(* CoDeSys 2.3.9.35 project: Exercício3.pro *)
(* Author: Altus *)
(* Libraries: DU35x.lib 7.7.11 15:59:13, Navigation.lib 15.7.11 10:06:00, SysLibTargetVisu.lib 26.11.08 09:53:28, Standard.lib 26.11.08 09:46:20, Iecsfc.lib 26.11.08 09:46:14, SYSLIBCALLBACK.LIB 26.11.08 09:53:30 *)

(* PLC configuration (modules and I/O channels)
Configuração do CP [Root] node -1, in %IB0 out %QB0
  Comunicação [Comunica] node 0, in %IB0 out %QB0
    COM1 [COM1] node 0, in %IB0 out %QB0 {BaudRate = 115200; Paridade = Sem Paridade; StopBits = 1 Stop Bit; Modem = Sem RTS/CTS; Delay = 5}
      MToolIEC [Codesys] node 0, in %IB0 out %QB0
    COM2 [COM2] node 1, in %IB0 out %QB0 {BaudRate = 115200; Paridade = Sem Paridade; StopBits = 1 Stop Bit; Modem = Sem RTS/CTS; Delay = 5}
      Desabilitada [Desabilitado485] node 0, in %IB0 out %QB0
  Barramento [Barramento] node 1, in %IB0 out %QB0
    Entradas [Entradas] node 0, in %IB0 out %QB0
      Entradas Digitais 0 [Entradas0] node 0, in %IW0 out %QB0
        I00 AT %IX0.0 [BitInput] I0.0
        I01 AT %IX0.1 [BitInput] I0.1
        I02 AT %IX0.2 [BitInput] I0.2
        I03 AT %IX0.3 [BitInput] I0.3
        I04 AT %IX0.4 [BitInput] I0.4
        I05 AT %IX0.5 [BitInput] I0.5
        I06 AT %IX0.6 [BitInput] I0.6
        I07 AT %IX0.7 [BitInput] I0.7
        I08 AT %IX0.8 [BitInput] I0.8
      Entradas Digitais 1 [Entradas1] node 0, in %IW1 out %QB0
        I10 AT %IX1.0 [BitInput] I1.0
        I11 AT %IX1.1 [BitInput] I1.1
        I12 AT %IX1.2 [BitInput] I1.2
        I13 AT %IX1.3 [BitInput] I1.3
        I14 AT %IX1.4 [BitInput] I1.4
        I15 AT %IX1.5 [BitInput] I1.5
        I16 AT %IX1.6 [BitInput] I1.6
        I17 AT %IX1.7 [BitInput] I1.7
        I18 AT %IX1.8 [BitInput] I1.8
      Entradas Digitais 2 [Entradas2] node 0, in %IW2 out %QB0
        I20 AT %IX2.0 [BitInput] I2.0
        I21 AT %IX2.1 [BitInput] I2.1
      Entradas Analógicas [EntradaAnalogica] node 0, in %IW4 out %QB0
        AI0 AT %IW4 [WordInput] AI0 {TipoAnalogica = Channel Disable; FiltroAnalogica = Filter 0 - AI=2ms  / AV=90ms; FundoEscala = 0}
        AI1 AT %IW5 [WordInput] AI1 {TipoAnalogica = Channel Disable; FiltroAnalogica = Filter 0 - AI=2ms  / AV=90ms; FundoEscala = 0}
        AI2 AT %IW6 [WordInput] AI2 {TipoAnalogica = Channel Disable; FiltroAnalogica = Filter 0 - AI=2ms  / AV=90ms; FundoEscala = 0}
        AI3 AT %IW7 [WordInput] AI3 {TipoAnalogica = Channel Disable; FiltroAnalogica = Filter 0 - AI=2ms  / AV=90ms; FundoEscala = 0}
      Entradas Rápidas [EntradasRapidas] node 1, in %IB16 out %QB0
        Bloco 0 [Bloco0] node 0, in %IB16 out %QB0
          Desabilitado [DesabilitadoBloco0] node 0, in %IB16 out %QB0
        Bloco 1 [Bloco1] node 1, in %IB16 out %QB0
          Desabilitado [DesabilitadoBloco1] node 0, in %IB16 out %QB0
        Entrada Configuravél Bloco 0 [EntradaConfiBloco0] node 2, in %IB16 out %QB0
          Contador 0 [EntradaConfContador0] node 0, in %IB16 out %QB0 {EntradaConfiguravelContador = Disable}
        Entrada Configuravél Bloco 1 [EntradaConfiBloco1] node 3, in %IB16 out %QB0
          Contador 2 [EntradaConfContador2] node 0, in %IB16 out %QB0 {EntradaConfiguravelContador = Disable}
    Saídas [Saidas] node 1, in %IB13 out %QB0
      Saídas Digitais 0 [Saidas0] node 0, in %IW0 out %QW0
        Q00 AT %QX0.0 [BitOutput] Q0.0
        Q01 AT %QX0.1 [BitOutput] Q0.1
        Q02 AT %QX0.2 [BitOutput] Q0.2
        Q03 AT %QX0.3 [BitOutput] Q0.3
        Q04 AT %QX0.4 [BitOutput] Q0.4
        Q05 AT %QX0.5 [BitOutput] Q0.5
        Q06 AT %QX0.6 [BitOutput] Q0.6
        Q07 AT %QX0.7 [BitOutput] Q0.7
      Saídas Digitais 1 [Saidas1] node 0, in %IW0 out %QW1
        Q10 AT %QX1.0 [BitOutput] Q1.0
        Q11 AT %QX1.1 [BitOutput] Q1.1
        Q12 AT %QX1.2 [BitOutput] Q1.2
        Q13 AT %QX1.3 [BitOutput] Q1.3
        Q14 AT %QX1.4 [BitOutput] Q1.4
        Q15 AT %QX1.5 [BitOutput] Q1.5
        Q16 AT %QX1.6 [BitOutput] Q1.6
        Q17 AT %QX1.7 [BitOutput] Q1.7
      Saídas Analógicas [SaidaAnalogica] node 0, in %IW0 out %QW3
        AO0 AT %QW3 [WordOutput] AO0 {TipoAnalogica = Channel Disable; FundoEscala = 0}
        AO1 AT %QW4 [WordOutput] AO1 {TipoAnalogica = Channel Disable; FundoEscala = 0}
      Saídas Rápidas [SaidasRapidas] node 1, in %IB0 out %QB10
        Saída Rápida 0 Desabilitada [DesabilitadoF0] node 0, in %IB0 out %QB10
        Saída Rápida 1 Desabilitada [DesabilitadoF1] node 1, in %IB0 out %QB10
      Saídas Comum de Contador [SaidasContador] node 2, in %IB0 out %QB10
        Saída do Bloco 0 Desabilitada [DesabilitadoSaidaBloco0] node 0, in %IB0 out %QB10
        Saída do Bloco 1 Desabilitada [DesabilitadoSaidaBloco1] node 1, in %IB0 out %QB10
  Eventos Externos [Eventos] node 2, in %IB13 out %QB6
    Evento Temporizado [TimerEvent] node 0, in %IB13 out %QB6 {Intervalo = 10}
*)

(* Task configuration *)
TASK PRINCIPAL (PRIORITY := 1, INTERVAL := T#1ms);
	PLC_PRG();
END_TASK
TASK NAVIGATION (PRIORITY := 1, INTERVAL := T#20ms);
	NAVEGA();
END_TASK
TASK VISUALIZATION (PRIORITY := 1, INTERVAL := T#500ms);
	MAINTARGETVISU_PAINT_CODE
END_TASK
TASK KEYBOARD_USAGE (PRIORITY := 1, INTERVAL := T#20ms);
	MAINTARGETVISU_INPUT_CODE
END_TASK

(* POU PLC_PRG, LD *)
(*Elabore um programa que produza uma rampa de tensão analógica para acionamento de um sistema partida e parada suaves de um motor (com um
sistema analógico com TCA785, por exemplo). Ao ser acionado um botão denominado LIGA no painel da IHM do CP, deve ser gerada uma rampa de 0V
a 10V na saída analógica, e de 10V a 0V ao ser acionado um botão denominado DESLIGA. O tempo de subida deve ser de 10s e tempo de descida de 
7s. Exiba o valor do percentual de potência na IHM. A rampa deve ter pelo menos 100 pontos de resolução. Prever o acionamento de uma saída 
digital no estado de potência zero e outra saída digital no estado de potência máxima. Exiba o valor de tensão de saída na IHM, de forma 
numérica e de forma gráfica (gráfico de tendência, por exemplo). Usar a escala apropriada (duas casa decimais) e com indicação de unidade.
*)

PROGRAM PLC_PRG
VAR
	LIG: BOOL;
	DES: BOOL;
	S1 AT %QX1.0: BOOL;
	S2 AT %QX1.1: BOOL := 1;
	AN AT %QW3: WORD;
	TS: TIME := T#10s;
	TD: TIME := T#7s;
	T1: TOF;
	T2: TOF;
	DESC: TIME;
	SUBI: TIME;
	BD1: F_TRIG;
	BD2: F_TRIG;
	BSS1: R_TRIG;
	BSS2: R_TRIG;
	BD: R_TRIG;
	BL: R_TRIG;
	M1: BOOL;
	M2: BOOL := 1;
	M3: BOOL;
	M4: BOOL;
	M5: BOOL;
	TR: WORD;
	SUBTR: REAL;
	SUBWORD: WORD;
	ANR: REAL;
	POT: REAL;
END_VAR
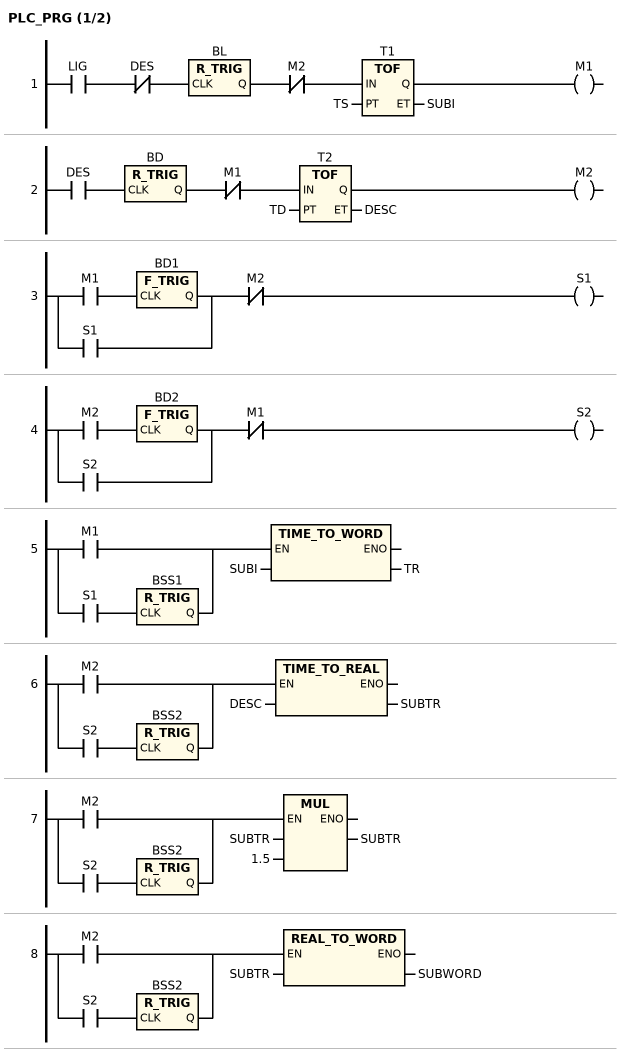
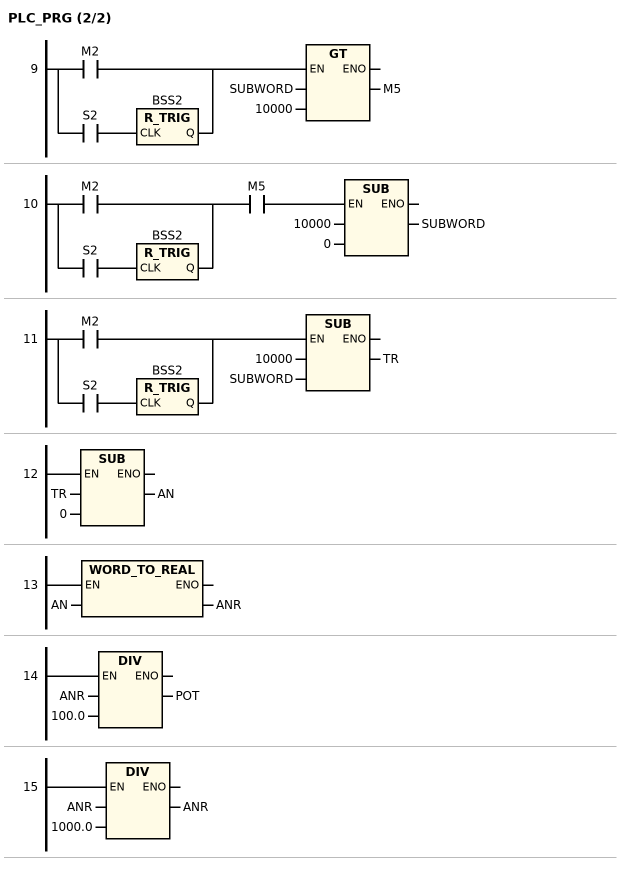
_LD_ (* Ladder Diagram *)
NETWORK 1
	[LIG] - [/DES] - BL:R_TRIG(CLK: *) - [/M2] - T1:TOF(IN: *, PT: TS, ET => SUBI) --- (M1)
NETWORK 2
	[DES] - BD:R_TRIG(CLK: *) - [/M1] - T2:TOF(IN: *, PT: TD, ET => DESC) --- (M2)
NETWORK 3
	{ [M1] - BD1:F_TRIG(CLK: *) | [S1] } - [/M2] --- (S1)
NETWORK 4
	{ [M2] - BD2:F_TRIG(CLK: *) | [S2] } - [/M1] --- (S2)
NETWORK 5
	{ [M1] | [S1] - BSS1:R_TRIG(CLK: *) }
		EN --- TIME_TO_WORD(SUBI) => TR
NETWORK 6
	{ [M2] | [S2] - BSS2:R_TRIG(CLK: *) }
		EN --- TIME_TO_REAL(DESC) => SUBTR
NETWORK 7
	{ [M2] | [S2] - BSS2:R_TRIG(CLK: *) }
		EN --- MUL(SUBTR, 1.5) => SUBTR
NETWORK 8
	{ [M2] | [S2] - BSS2:R_TRIG(CLK: *) }
		EN --- REAL_TO_WORD(SUBTR) => SUBWORD
NETWORK 9
	{ [M2] | [S2] - BSS2:R_TRIG(CLK: *) }
		EN --- GT(SUBWORD, 10000) => M5
NETWORK 10
	{ [M2] | [S2] - BSS2:R_TRIG(CLK: *) } - [M5]
		EN --- SUB(10000, 0) => SUBWORD
NETWORK 11
	{ [M2] | [S2] - BSS2:R_TRIG(CLK: *) }
		EN --- SUB(10000, SUBWORD) => TR
NETWORK 12
	*
		EN --- SUB(TR, 0) => AN
NETWORK 13
	*
		EN --- WORD_TO_REAL(AN) => ANR
NETWORK 14
	*
		EN --- DIV(ANR, 100.0) => POT
NETWORK 15
	*
		EN --- DIV(ANR, 1000.0) => ANR
_END_LD_
(* the same logic as Structured Text *)
(* Network 1 *)
BL(CLK := LIG AND NOT DES);
T1(IN := BL.Q AND NOT M2, PT := TS);
SUBI := T1.ET;
M1 := T1.Q;
(* Network 2 *)
BD(CLK := DES);
T2(IN := BD.Q AND NOT M1, PT := TD);
DESC := T2.ET;
M2 := T2.Q;
(* Network 3 *)
BD1(CLK := M1);
S1 := (BD1.Q OR S1) AND NOT M2;
(* Network 4 *)
BD2(CLK := M2);
S2 := (BD2.Q OR S2) AND NOT M1;
(* Network 5 *)
BSS1(CLK := S1);
IF M1 OR BSS1.Q THEN
	TR := TIME_TO_WORD(SUBI);
END_IF;
(* Network 6 *)
BSS2(CLK := S2);
IF M2 OR BSS2.Q THEN
	SUBTR := TIME_TO_REAL(DESC);
END_IF;
(* Network 7 *)
BSS2(CLK := S2);
IF M2 OR BSS2.Q THEN
	SUBTR := SUBTR * 1.5;
END_IF;
(* Network 8 *)
BSS2(CLK := S2);
IF M2 OR BSS2.Q THEN
	SUBWORD := REAL_TO_WORD(SUBTR);
END_IF;
(* Network 9 *)
BSS2(CLK := S2);
IF M2 OR BSS2.Q THEN
	M5 := SUBWORD > 10000;
END_IF;
(* Network 10 *)
BSS2(CLK := S2);
IF (M2 OR BSS2.Q) AND M5 THEN
	SUBWORD := 10000 - 0;
END_IF;
(* Network 11 *)
BSS2(CLK := S2);
IF M2 OR BSS2.Q THEN
	TR := 10000 - SUBWORD;
END_IF;
(* Network 12 *)
AN := TR - 0;
(* Network 13 *)
ANR := WORD_TO_REAL(AN);
(* Network 14 *)
POT := ANR / 100.0;
(* Network 15 *)
ANR := ANR / 1000.0;
END_PROGRAM

(* POU NAVEGA, ST *)
PROGRAM NAVEGA
VAR
	ControleTelas : NAVIGATION;
	ListaTelas 	: ARRAY [0..30] OF STRING(10);
END_VAR
(* Adiciona a tela MAIN como tela principal *)
ListaTelas[0] := 'MAIN';

(* Ativa o controle automático de navegação somente pelo teclado *)
ControleTelas(ENABLE_UPDW := FALSE, VISU_LIST := ListaTelas, UP := FALSE , DOWN := FALSE);
END_PROGRAM

(* Visualisation MAIN
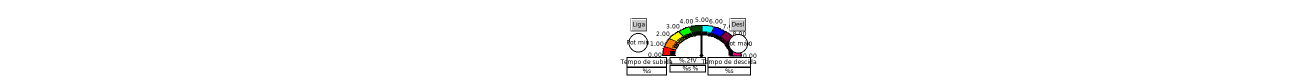
group at (20,0)-(129,45)
  rectangle at (0,0)-(1,1): text "{ExtendedElement},Visu\ElementDLL.ete,0,@Zeigerinstrument,109,180,0,3,0,0,0,0,PLC_PRG.ANR,,%.2f,0,1,1,0.1,1,0,10,0,0,0,0,0,0,0,-5,40,400,Arial,1,10,0,1,255,0,0,1,2,255,128,0,2,3,255,255,0,3,4,0,255,0,4,5,0,64,0,5,6,0,255,255,6,7,0,0,255,7,8,128,0,64,8,9,64,0,64,9,10,255,0,128,"
  rectangle at (4,51)-(14,57): text "0.00"
  rectangle at (6,37)-(16,43): text "1.00"
  rectangle at (12,24)-(22,30): text "2.00"
  rectangle at (22,14)-(32,20): text "3.00"
  rectangle at (35,8)-(45,14): text "4.00"
  rectangle at (50,6)-(60,12): text "5.00"
  rectangle at (64,8)-(74,14): text "6.00"
  rectangle at (77,14)-(87,20): text "7.00"
  rectangle at (87,24)-(97,30): text "8.00"
  rectangle at (93,37)-(103,43): text "9.00"
  rectangle at (94,52)-(107,58): text "10.00"
  polygon at (54,29)-(55,55): angle ((PLC_PRG.ANR * 1.0)-5) * 18
rectangle at (44,44)-(80,51): text "%.2fV"; shows PLC_PRG.ANR
rectangle at (1,44)-(41,54): text "Tempo de subida"
rectangle at (82,44)-(125,54): text "Tempo de descida"
rectangle at (1,54)-(41,62): text "%s"; shows PLC_PRG.SUBI
rectangle at (82,54)-(125,62): text "%s"; shows PLC_PRG.DESC
button at (5,5)-(21,18): text "Liga"; toggles PLC_PRG.LIG
button at (104,5)-(120,18): text "Desl"; toggles PLC_PRG.DES
rectangle at (44,52)-(80,59): text "%s"; shows PLC_PRG.POT
ellipse at (103,21)-(122,40): text "Pot máx"; alarm colour if PLC_PRG.S1
rectangle at (60,52)-(79,59): text "%"
ellipse at (3,20)-(22,39): text "Pot min"; alarm colour if PLC_PRG.S2
114 more shapes without text or variables
*)
